(* PLC project mbNewproject.project, Prosoft-Systems Ltd. Astra.IDE Astra.IDE V1.7.0.0 *)
(* stored: creationDateTime 2023-08-18T15:56:28.48287, modificationDateTime 2023-08-18T15:48:29.8985699 *)

PROGRAM MbControl

            
            ST CODE
		
          
END_PROGRAM
